FUNCTION_BLOCK CONCATENATE_REALS
  {SET_ATTRIBUTE(OpcUa, SERVICE)}
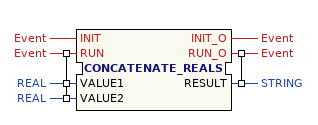
  EVENT_INPUT
    INIT;
    RUN WITH VALUE1, VALUE2;
  END_EVENT
  EVENT_OUTPUT
    INIT_O;
    RUN_O WITH RESULT;
  END_EVENT
  VAR_INPUT
    VALUE1 : REAL; {SET_ATTRIBUTE(OpcUa, Variable.RUN)}
    VALUE2 : REAL; {SET_ATTRIBUTE(OpcUa, Variable.RUN)}
  END_VAR
  VAR_OUTPUT
    RESULT : STRING; {SET_ATTRIBUTE(OpcUa, Variable.RUN)}
  END_VAR
END_FUNCTION_BLOCK
